Staubli VAL3: SendSpeed.pgx

public program SendSpeed(num x_nSpeed (dimensions=1))
begin
  //2014.3.24 设置机器人速度到O2_aNull
  x_nSpeed=max(0,x_nSpeed)
  aioSet(aAio["O2_aNull"],x_nSpeed)



end
